TYPE ST_HmiAxisManager :
STRUCT
	// axis selection
	eAxis : E_Axis;
	// enable hmi axis mgr
	bEnableAxisMgr : BOOL;

	// global axis manager
	stAxisManager	: REFERENCE TO ST_AxisManager;
END_STRUCT
END_TYPE

(* stored: Version 1.1.0.1, ProductVersion 3.1.4024.12
   DUT ST_HmiAxisManager: Id {192e7d07-1b34-48b3-9aa4-33e9c884ff60} *)
